// TIA Portal V19 export
DATA_BLOCK "DI_FU_Hub_links"   // DB182
// stored: AutoNumber false, InstanceOfName FB_FU_OUT_TW, InstanceOfType FB
"FB_FU_OUT_TW"
   // VAR_INPUT
   //    Req_High : Bool;
   //    Req_Low : Bool;
   // END_VAR
   // VAR_IN_OUT
   //    Reglersperre : Bool;
   //    Freigabe_Stopp : Bool;
   //    Freigabe_Halt : Bool;
   //    Break_ok : Bool;
   //    SollSpeed : Int;
   //    Ist_Speed : Int;
   //    PAW_Speed : Int;
   //    PEW_Speed : Int;
   // END_VAR
   // VAR RETAIN
   //    maxSpeed : Real;
   //    Faktor { ExternalAccessible := 'False'; ExternalVisible := 'False'; ExternalWritable := 'False'} : Real;
   //    minSpeed : Int;
   // END_VAR
BEGIN
END_DATA_BLOCK
